// TwinCAT 3 PLC project M3K2
// ProgramVersion: 3.1.4022.7
// libraries:
//   LCLS General, * (SLAC)
//   lcls-twincat-motion, * (SLAC)
//   Tc2_MC2, * (Beckhoff Automation GmbH)
//   Tc2_Standard, * (Beckhoff Automation GmbH)
//   Tc2_System, * (Beckhoff Automation GmbH)
//   Tc3_Module, * (Beckhoff Automation GmbH)
// project tree:
//   / PlcTask.TcTTO (not stored)
//   POUs/ FB_MotionStageStats.TcPOU, FB_PAT.TcPOU (not stored), Main.TcPOU
// real-time tasks:
//   TASK PlcTask: cycle T#10ms, priority 20, ADS port 350
// motion (NC):
//   TASK NC-Task 1 SAF: cycle T#2ms, priority 4, ADS port 501
//   TASK NC-Task 1 SVB: cycle T#10ms, priority 8, ADS port 511
//   AXIS M4K2 X (id 1)
//     Dynamic: AccelerationMaximum=100, DecelerationMaximum=100, Acceleration=100, Deceleration=100, DelayTime=0.008
//     Velo: Maximum=20
//     OtherSettings: AllowMotionCmdToSlave=true
//     encoder EncType=29
//       EncPara: ScaleFactorNumerator=5e-06, Offset=-29.51, MaxCount=#xffffffff, ReferenceSystem=1
//         Inc: RefSoftSyncMask=#x00000000
//     drive DrvType=24
//       DrvPara: Inverse=true
//         Analog: VeloReferenz=20, ScaleFactorActTorque=0.1
//         TimeComp: TaskDelayCycles=1
//     controller CtrType=1
//       CtrPara: PriorControlFactor=1
//         PosDiffControl: Range=0.1
//         Observer: BandWidth=20
//   AXIS M4K2 Y (id 2)
//     Dynamic: AccelerationMaximum=10, DecelerationMaximum=10, Acceleration=10, Deceleration=10, Jerk=15, DelayTime=0.008
//     Velo: Maximum=1.25
//     OtherSettings: AllowMotionCmdToSlave=true
//     encoder EncType=29
//       EncPara: ScaleFactorNumerator=5e-06, Offset=-30, MaxCount=#xffffffff, ReferenceSystem=1
//         Inc: RefSoftSyncMask=#x00000000
//     drive DrvType=24
//       DrvPara: Inverse=true
//         Analog: VeloReferenz=1.25, ScaleFactorActTorque=0.1
//         TimeComp: TaskDelayCycles=1
//     controller CtrType=1
//       CtrPara: PriorControlFactor=1
//         PosDiffControl: Range=0.1
//         Observer: BandWidth=20
//   AXIS M4K2 rX (id 3)
//     General: UnitName=urad
//     Dynamic: AccelerationMaximum=200, DecelerationMaximum=200, Acceleration=200, Deceleration=200, DelayTime=0.008
//     Velo: Maximum=20
//     OtherSettings: AllowMotionCmdToSlave=true
//     encoder EncType=29
//       EncPara: ScaleFactorNumerator=0.002571, Offset=-836.5, MaxCount=#x00061a80, ReferenceSystem=1
//         Inc: RefSoftSyncMask=#x00000000
//     drive DrvType=24
//       DrvPara: Inverse=true
//         Analog: VeloReferenz=20, ScaleFactorActTorque=0.1
//         TimeComp: TaskDelayCycles=1
//     controller CtrType=1
//       CtrPara: PriorControlFactor=1
//         PosDiffControl: Range=10
//         PID: PosKp=5, PosExtKp=1, DeadBandPosition=0.01
//         Observer: BandWidth=20
// I/O:
//   DEVICE Device 1 (EtherCAT), AmsNetId 192.168.0.19.2.1
//     Term 1 (EK1100) [EK1100 EtherCAT Coupler (2A E-Bus)]
//       Term 2 (EL5042) [EL5042 2Ch. BiSS-C Encoder]
//       Term 3 (EL5042) [EL5042 2Ch. BiSS-C Encoder]
//       Term 4 (EL9221-5000) [EL9221-5000 Overcurrent protection 24V DC, 1Ch., max. 10A, adjustable]
//       M3K2 X [EL7041-0052 1Ch. Stepper motor output stage (50V, 5A)]
//       M3K2 Y [EL7041-0052 1Ch. Stepper motor output stage (50V, 5A)]
//       M3K2 rX [EL7041-0052 1Ch. Stepper motor output stage (50V, 5A)]
//       STO (EL1004) [EL1004 4Ch. Dig. Input 24V, 3ms]
//       Term 9 (EL9011) [EL9011 End Terminal]
// variable links:
//   (this object) <-> Device 1 (EtherCAT)/Term 1 (EK1100)/M4K2 X
//     Drive/Inputs/In/nState1 @bit 3 <-> STM Status/Status/Error
//     Drive/Inputs/In/nState1 @bit 5 <-> STM Status/Status/Moving negative
//     Drive/Inputs/In/nState1 @bit 4 <-> STM Status/Status/Moving positive
//     Drive/Inputs/In/nState1 @bit 1 <-> STM Status/Status/Ready
//     Drive/Inputs/In/nState1 <-> STM Status/Status/Ready to enable
//     Drive/Inputs/In/nState1 @bit 6 <-> STM Status/Status/Torque reduced
//     Drive/Inputs/In/nState1 @bit 2 <-> STM Status/Status/Warning
//     Drive/Inputs/In/nState2 @bit 3 <-> STM Status/Status/Digital input 1
//     Drive/Inputs/In/nState2 @bit 4 <-> STM Status/Status/Digital input 2
//     Drive/Inputs/In/nState2 @bit 5 <-> STM Status/Status/Sync error
//     Drive/Inputs/In/nState2 @bit 7 <-> STM Status/Status/TxPDO Toggle
//     Drive/Inputs/In/nState4 @bit 1 <-> WcState/InputToggle
//     Drive/Inputs/In/nState4 <-> WcState/WcState
//     Drive/Outputs/Out/nCtrl1 <-> STM Control/Control/Enable
//     Drive/Outputs/Out/nCtrl1 @bit 2 <-> STM Control/Control/Reduce torque
//     Drive/Outputs/Out/nCtrl1 @bit 1 <-> STM Control/Control/Reset
//     Drive/Outputs/Out/nDataOut2[0] <-> STM Velocity/Velocity
//   (this object) <-> Device 1 (EtherCAT)/Term 1 (EK1100)/Term 2 (EL5042)
//     Enc/Inputs/In/nComState @bit 1 <-> WcState/InputToggle
//     Enc/Inputs/In/nComState <-> WcState/WcState
//     Enc/Inputs/In/nDataIn1 <-> FB Inputs Channel 1/Position
//     Enc/Inputs/In/nDataIn1 <-> FB Inputs Channel 2/Position
//     Enc/Inputs/In/nState1 @bit 12 <-> FB Inputs Channel 1/Status/Diag
//     Enc/Inputs/In/nState1 @bit 12 <-> FB Inputs Channel 2/Status/Diag
//     Enc/Inputs/In/nState1 @bit 1 <-> FB Inputs Channel 1/Status/Error
//     Enc/Inputs/In/nState1 @bit 1 <-> FB Inputs Channel 2/Status/Error
//     Enc/Inputs/In/nState1 @bit 14 <-> FB Inputs Channel 1/Status/Input cycle counter
//     Enc/Inputs/In/nState1 @bit 14 <-> FB Inputs Channel 2/Status/Input cycle counter
//     Enc/Inputs/In/nState1 @bit 2 <-> FB Inputs Channel 1/Status/Ready
//     Enc/Inputs/In/nState1 @bit 2 <-> FB Inputs Channel 2/Status/Ready
//     Enc/Inputs/In/nState1 @bit 13 <-> FB Inputs Channel 1/Status/TxPDO State
//     Enc/Inputs/In/nState1 @bit 13 <-> FB Inputs Channel 2/Status/TxPDO State
//     Enc/Inputs/In/nState1 <-> FB Inputs Channel 1/Status/Warning
//     Enc/Inputs/In/nState1 <-> FB Inputs Channel 2/Status/Warning
//   (this object) <-> Device 1 (EtherCAT)/Term 1 (EK1100)/M4K2 Y
//     Drive/Inputs/In/nState1 @bit 3 <-> STM Status/Status/Error
//     Drive/Inputs/In/nState1 @bit 5 <-> STM Status/Status/Moving negative
//     Drive/Inputs/In/nState1 @bit 4 <-> STM Status/Status/Moving positive
//     Drive/Inputs/In/nState1 @bit 1 <-> STM Status/Status/Ready
//     Drive/Inputs/In/nState1 <-> STM Status/Status/Ready to enable
//     Drive/Inputs/In/nState1 @bit 6 <-> STM Status/Status/Torque reduced
//     Drive/Inputs/In/nState1 @bit 2 <-> STM Status/Status/Warning
//     Drive/Inputs/In/nState2 @bit 3 <-> STM Status/Status/Digital input 1
//     Drive/Inputs/In/nState2 @bit 4 <-> STM Status/Status/Digital input 2
//     Drive/Inputs/In/nState2 @bit 5 <-> STM Status/Status/Sync error
//     Drive/Inputs/In/nState2 @bit 7 <-> STM Status/Status/TxPDO Toggle
//     Drive/Inputs/In/nState4 @bit 1 <-> WcState/InputToggle
//     Drive/Inputs/In/nState4 <-> WcState/WcState
//     Drive/Outputs/Out/nCtrl1 <-> STM Control/Control/Enable
//     Drive/Outputs/Out/nCtrl1 @bit 2 <-> STM Control/Control/Reduce torque
//     Drive/Outputs/Out/nCtrl1 @bit 1 <-> STM Control/Control/Reset
//     Drive/Outputs/Out/nDataOut2[0] <-> STM Velocity/Velocity
//   (this object) <-> Device 1 (EtherCAT)/Term 1 (EK1100)/M4K2 rX
//     Drive/Inputs/In/nState1 @bit 3 <-> STM Status/Status/Error
//     Drive/Inputs/In/nState1 @bit 5 <-> STM Status/Status/Moving negative
//     Drive/Inputs/In/nState1 @bit 4 <-> STM Status/Status/Moving positive
//     Drive/Inputs/In/nState1 @bit 1 <-> STM Status/Status/Ready
//     Drive/Inputs/In/nState1 <-> STM Status/Status/Ready to enable
//     Drive/Inputs/In/nState1 @bit 6 <-> STM Status/Status/Torque reduced
//     Drive/Inputs/In/nState1 @bit 2 <-> STM Status/Status/Warning
//     Drive/Inputs/In/nState2 @bit 3 <-> STM Status/Status/Digital input 1
//     Drive/Inputs/In/nState2 @bit 4 <-> STM Status/Status/Digital input 2
//     Drive/Inputs/In/nState2 @bit 5 <-> STM Status/Status/Sync error
//     Drive/Inputs/In/nState2 @bit 7 <-> STM Status/Status/TxPDO Toggle
//     Drive/Inputs/In/nState4 @bit 1 <-> WcState/InputToggle
//     Drive/Inputs/In/nState4 <-> WcState/WcState
//     Drive/Outputs/Out/nCtrl1 <-> STM Control/Control/Enable
//     Drive/Outputs/Out/nCtrl1 @bit 2 <-> STM Control/Control/Reduce torque
//     Drive/Outputs/Out/nCtrl1 @bit 1 <-> STM Control/Control/Reset
//     Drive/Outputs/Out/nDataOut2[0] <-> STM Velocity/Velocity
//   (this object) <-> Device 1 (EtherCAT)/Term 1 (EK1100)/Term 3 (EL5042)
//     Enc/Inputs/In/nComState @bit 1 <-> WcState/InputToggle
//     Enc/Inputs/In/nComState <-> WcState/WcState
//     Enc/Inputs/In/nDataIn1 <-> FB Inputs Channel 1/Position
//     Enc/Inputs/In/nState1 @bit 12 <-> FB Inputs Channel 1/Status/Diag
//     Enc/Inputs/In/nState1 @bit 1 <-> FB Inputs Channel 1/Status/Error
//     Enc/Inputs/In/nState1 @bit 14 <-> FB Inputs Channel 1/Status/Input cycle counter
//     Enc/Inputs/In/nState1 @bit 2 <-> FB Inputs Channel 1/Status/Ready
//     Enc/Inputs/In/nState1 @bit 13 <-> FB Inputs Channel 1/Status/TxPDO State
//     Enc/Inputs/In/nState1 <-> FB Inputs Channel 1/Status/Warning
//   M3K2 Instance <-> Device 1 (EtherCAT)/Term 1 (EK1100)/M3K2 X
//     PlcTask Inputs/Main.M1.bLimitBackwardEnable <-> STM Status/Status/Digital input 2
//     PlcTask Inputs/Main.M1.bLimitForwardEnable <-> STM Status/Status/Digital input 1
//   M3K2 Instance <-> Device 1 (EtherCAT)/Term 1 (EK1100)/M3K2 Y
//     PlcTask Inputs/Main.M2.bLimitBackwardEnable <-> STM Status/Status/Digital input 2
//     PlcTask Inputs/Main.M2.bLimitForwardEnable <-> STM Status/Status/Digital input 1
//   M3K2 Instance <-> Device 1 (EtherCAT)/Term 1 (EK1100)/M3K2 rX
//     PlcTask Inputs/Main.M3.bLimitBackwardEnable <-> STM Status/Status/Digital input 2
//     PlcTask Inputs/Main.M3.bLimitForwardEnable <-> STM Status/Status/Digital input 1
//   M3K2 Instance <-> Device 1 (EtherCAT)/Term 1 (EK1100)/STO (EL1004)
//     PlcTask Inputs/Main.bSTOEnable1 <-> Channel 1/Input
//     PlcTask Inputs/Main.bSTOEnable2 <-> Channel 2/Input
//   M3K2 Instance <-> NC-Task 1 SAF/Axes/M2K2 X
//     PlcTask Inputs/Main.M1.Axis.NcToPlc <-> Outputs/ToPlc
//     PlcTask Outputs/Main.M1.Axis.PlcToNc <-> Inputs/FromPlc
//   M3K2 Instance <-> NC-Task 1 SAF/Axes/M2K2 Y
//     PlcTask Inputs/Main.M2.Axis.NcToPlc <-> Outputs/ToPlc
//     PlcTask Outputs/Main.M2.Axis.PlcToNc <-> Inputs/FromPlc
//   M3K2 Instance <-> NC-Task 1 SAF/Axes/M2K2 rX
//     PlcTask Inputs/Main.M3.Axis.NcToPlc <-> Outputs/ToPlc
//     PlcTask Outputs/Main.M3.Axis.PlcToNc <-> Inputs/FromPlc

// ---- POUs/FB_MotionStageStats.TcPOU
FUNCTION_BLOCK FB_MotionStageStats EXTENDS FB_BasicStats
VAR_INPUT
    Axis : DUT_MotionStage;
END_VAR
VAR_OUTPUT
END_VAR
VAR
    aActPos : ARRAY [0..ARRAY_SIZE] OF LREAL;
    idx: UINT;
END_VAR
VAR CONSTANT
    ARRAY_SIZE : UINT := 500;
END_VAR


aActPos[idx] := Axis.Axis.NcToPlc.ActPos;

idx := (idx + 1) MOD ARRAY_SIZE;

SUPER^(aSignal:=aActPos, bAlwaysCalc:=NOT bReset);

END_FUNCTION_BLOCK

// ---- POUs/Main.TcPOU
PROGRAM Main
VAR
    {attribute 'TcLinkTo' := '.bLimitForwardEnable:=TIIB[M2K2 X]^STM Status^Status^Digital input 1;
                              .bLimitBackwardEnable:=TIIB[M2K2 X]^STM Status^Status^Digital input 2'}
    M1 : DUT_MotionStage := (nEnableMode:=ENUM_StageEnableMode.DURING_MOTION, bPowerSelf:=TRUE);
    fbMotionStageM1 : FB_MotionStage;
    {attribute 'TcLinkTo' := '.bLimitForwardEnable:=TIIB[M2K2 Y]^STM Status^Status^Digital input 1;
                              .bLimitBackwardEnable:=TIIB[M2K2 Y]^STM Status^Status^Digital input 2'}
    M2 : DUT_MotionStage := (nEnableMode:=ENUM_StageEnableMode.DURING_MOTION, bPowerSelf:=TRUE);
    fbMotionStageM2 : FB_MotionStage;
    {attribute 'TcLinkTo' := '.bLimitForwardEnable:=TIIB[M2K2 rX]^STM Status^Status^Digital input 1;
                              .bLimitBackwardEnable:=TIIB[M2K2 rX]^STM Status^Status^Digital input 2'}
    M3 : DUT_MotionStage := (nEnableMode:=ENUM_StageEnableMode.DURING_MOTION, bPowerSelf:=TRUE);
    fbMotionStageM3 : FB_MotionStage;


    fbStepSizeTest_M2K2X : FB_MicroStepCountTest := (
        fStepSize := 0.00015625,
        nSteps := 1000,
        fMicroStep := 0.00015625,
        fVelocity := 1,
        tSettleTime := T#1S);

    fbStepSizeTest_M2K2Y : FB_MicroStepCountTest := (
        fStepSize := 0.0097656,
        nSteps := 1000,
        fMicroStep := 0.0097656,
        fVelocity := 0.5,
        tSettleTime := T#1S);

    fbStepSizeTest_M2K2rX : FB_MicroStepCountTest := (
        fStepSize := 0.0013021,
        nSteps := 1000,
        fMicroStep := 0.0013021,
        fVelocity := 10,
        tSettleTime := T#1S);

    fbM1Stats : FB_MotionStageStats;
    fbM2Stats : FB_MotionStageStats;
    fbM3Stats : FB_MotionStageStats;

    {attribute 'TcLinkTo' := 'TIID^Device 1 (EtherCAT)^Term 1 (EK1100)^STO (EL1004)^Channel 1^Input'}
    bSTOEnable1 AT %I* : BOOL;
    {attribute 'TcLinkTo' := 'TIID^Device 1 (EtherCAT)^Term 1 (EK1100)^STO (EL1004)^Channel 2^Input'}
    bSTOEnable2 AT %I* : BOOL;

    END_VAR


M1.bHardwareEnable := bSTOEnable1 AND bSTOEnable2;
M2.bHardwareEnable := bSTOEnable1 AND bSTOEnable2;
M3.bHardwareEnable := bSTOEnable1 AND bSTOEnable2;

fbMotionStageM1(stMotionStage:=M1);
fbMotionStageM2(stMotionStage:=M2);
fbMotionStageM3(stMotionStage:=M3);

fbM1Stats(Axis:=M1);
fbM2Stats(Axis:=M2);
fbM3Stats(Axis:=M3);

fbStepSizeTest_M2K2X(Axis:=M1.Axis);
fbStepSizeTest_M2K2Y(Axis:=M2.Axis);
fbStepSizeTest_M2K2rX(Axis:=M3.Axis);

END_PROGRAM
